TYPE ST_ProductData :
STRUCT
	
	nSerial				: UDINT;
	bInitRun			: BOOL;
	nDestinationProcess	: UINT;
	nPriority			: UINT;
	

END_STRUCT
END_TYPE

(* stored: Version 1.1.0.1, ProductVersion 3.1.4024.9
   DUT ST_ProductData: Id {5359bd88-833e-4f3c-b85b-bef29679fc9d} *)
